PROGRAM registerProc21
VAR
	i: INT;
	tempo: ton;
	state: INT;
	user: string;
END_VAR

tempo();

CASE state OF
	
0:
IF gvl_p.etapa_process[2] = 'Secagem' or gvl_p.etapa_process[2] = 'T1' THEN
	state:=10;
	tempo(in:=TRUE, pt:=T#30M);
ELSE
	state:=0;
END_IF

10:
IF tempo.Q THEN
	state:= 20;
IF i=1 THEN
gvl.permanencia[3]:= gvl.permanencia[3]+tempo.PT;
user:= main.sDB_Operador;
END_IF
IF gvl_p.aPositionsE021[i].reator THEN
	gvl.sReator:= 'SIM';
	else
		gvl.sReator:= 'NÃO';
END_IF
IF gvl_p.aPositionsE021[i].FP = 1 THEN
	gvl.sFp:= 'NORMAL';
	ELSIF gvl_p.aPositionsE021[i].FP = 2 THEN
		gvl.sFp:= 'REDUZIDO';
END_IF
IF gvl_p.aPositionsE021[i].isolamento = 1 THEN
	gvl.sIso:= '15';
	ELSIF gvl_p.aPositionsE021[i].isolamento = 2 THEN
		gvl.sIso:= '24';
		ELSIF gvl_p.aPositionsE021[i].isolamento = 3 THEN
			gvl.sIso:= '36';
END_IF
IF gvl_p.arrStatusEstufas[2].start THEN
	gvl.sAuto:= 'Auto';
	ELSIF gvl_p.arrStatusEstufas[2].startManual THEN
		gvl.sAuto:= 'Manu';
END_IF

gvl.sCmdInsertProc:= 'INSERT INTO [dbo].[ProcessTable21] ([data],[hora],[auto],[user],[pos],[OF],[lote],[class],[pot],[isola],[fPot],[reator],[TIME],[temp])
	VALUES ($'$',$'$',$'$',$'$',$'$',$'$',$'$',,,$'$',$'$',$'$',$'$',)';
gvl.sCmdInsertProc:= insert(gvl.sCmdInsertProc,REAL_TO_STRING(gvl.zona1atual_021),180);
gvl.sCmdInsertProc:= insert(gvl.sCmdInsertProc,TIME_TO_STRING(gvl.permanencia[3]),178);
gvl.sCmdInsertProc:= insert(gvl.sCmdInsertProc,gvl.sReator,175);
gvl.sCmdInsertProc:= insert(gvl.sCmdInsertProc,gvl.sFp,172);
gvl.sCmdInsertProc:= insert(gvl.sCmdInsertProc,gvl.sIso,169);
gvl.sCmdInsertProc:= insert(gvl.sCmdInsertProc,REAL_TO_STRING(gvl_p.aPositionsE021[i].pot),167);
gvl.sCmdInsertProc:= insert(gvl.sCmdInsertProc,REAL_TO_STRING(gvl_p.aPositionsE021[i].class),166);
gvl.sCmdInsertProc:= insert(gvl.sCmdInsertProc,gvl_p.aPositionsE021[i].lote,164);
gvl.sCmdInsertProc:= insert(gvl.sCmdInsertProc,gvl_p.aPositionsE021[i].numOF,161);
gvl.sCmdInsertProc:= insert(gvl.sCmdInsertProc,INT_TO_STRING(i),158);
gvl.sCmdInsertProc:= insert(gvl.sCmdInsertProc,user,155);
gvl.sCmdInsertProc:= insert(gvl.sCmdInsertProc,gvl.sAuto,152);
gvl.sCmdInsertProc:= insert(gvl.sCmdInsertProc,gvl.sSystemTime,149);
gvl.sCmdInsertProc:= insert(gvl.sCmdInsertProc,gvl.sSystemDate,146);

gvl.bInsertProc:= TRUE;
ELSE
	state:=10;
END_IF

20:
IF i<=24 AND NOT main.bBusyInsertProc THEN
	state:=10;
	i:=i+1;
ELSIF i=24 THEN
	state:=0;
	i:=1;
	tempo(in:=FALSE);
ELSE
	state:=20;
END_IF

END_CASE

END_PROGRAM

(* stored: Version 1.1.0.1, ProductVersion 3.1.4024.12
   POU registerProc21: Id {4a2f36ca-8d9a-4834-8de6-869c3420b249}, SpecialFunc None *)
